PROGRAM MAIN
VAR
	RuntimeDuration	: STRING;
	TempRuntimeDur	: TIME;
	RuntimeTimer	: TON;
	CurrentSysTime	: ULINT;

	bAllDone		: BOOL;
	bStopSequence	: BOOL;
	HMI_StopCmd		: BOOL;
	
	nCase 		: INT;
	nMoveState		: ARRAY[1..nMoverCount] OF INT;
	

	
	nForCounter: UDINT;
	M,N,T,Tr : UINT;
//	slowDynamics: DynamicConstraint_PathXY;
	haltDynamics : DynamicConstraint_PathXY;
	stopAndWait : ARRAY[1..GVL_Mc.nMoverCount] OF TON; 
	waitForGapParkPos: LREAL := 3500;
	// Magnet
	MagnetValue AT%Q*: INT;
	MagnetFdbkValue AT%I* : INT;
	bMagnetOn : BOOL;
	MagnetOnManHMICmd 	: BOOL;
	tMagnetOnTime	: TIME := T#3S;

	Init : BOOL ; 	
	
	IsMoverCommandedInShortcut: BOOL;
	IsMoverInBlockingArea: BOOL;
	nActStopPos: UINT := 1;
	Fp_error : R_Trig;

	Switch : BOOL;
	WithoutSwitch : BOOL := TRUE;
	SwtichOnly: BOOL;
	
	MoverStop 	AT%I* :BOOL;
	MoverStopDone AT%Q*		: BOOL;
	Info 		AT%Q*: BOOL;
	Operating	AT%Q*: BOOL;
	Process		AT%Q*: BOOL;
	Fault		AT%Q*: BOOL;
	Emergency	AT%Q*: BOOL;
	
	Voltage1 AT%I*: UDINT;
	Voltage2 AT%I*: UDINT;
	
	
	TcRestart : TC_Restart;
	Restart : BOOL;
	busy : BOOL;
	rt_InitStart : R_TRIG;
	rt_InitStop : R_TRIG;
	bStartSequence: BOOL;
	
	FP_Counter : r_trig;
	Switchcounter : DINT;
	test : LREAL;
	Horntimer : tp; 
	R_trigHorn : R_trig;
	
	TestPowerMat : BOOL := TRUE;
	StopTime : TIME := T#1S;
	StopTimer :ARRAY[1..nMoverCount] OF ton;
	StartTimer :ARRAY[1..nMoverCount] OF BOOL;
	
	
	MoverPos :ARRAY[1..nMoverCount] OF PositionXYC;
	ArcLength :ARRAY[1..nMoverCount] OF LREAL;
	TrackPos :ARRAY[1..nMoverCount] OF ARRAY[1..nMoverCount] OF PositionXYC;
	
	//searchGap : F_SearchTheBigTrackForAHole; 
	aMoverTrack : ARRAY[1..nMoverCount] OF Global.OTCID;
	FirstMoverTrackPos : LREAL;
	MoverGap : LREAL;
	FTrigTrackCount : F_Trig;
	MoverNo  : UDINT;
	stMoverConfigSlow	: ST_MoverConfig;
	stMoverConfigNormal : ST_MoverConfig;
	stMoverConfigFast  : ST_MoverConfig;
	stMoverCfgAggressive : ST_MoverConfig;
	stMoverCfgHalt : ST_MoverConfig;
	
	stMergeConfig		 : ST_MergeConfig;
	SwitchConfig		 : ST_SwitchConfig;
	
	SwitchStatus 		  : ST_SwitchStatus;

	ModuleState1 AT%I*: E_EcState;
	ModuleState2 AT%I*: E_EcState;
	ModuleState3 AT%I*: ARRAY[0..2] OF E_EcState;
	
	MessageTrigger : ARRAY[1..20] OF R_trig;
	
	//========= Merge =========================================
	
	SwitchParkPos : LREAL := 3500;
	nextMoverForSwitch: UDINT :=1;
	moverInSwitchDoNotSendAnother: BOOL;
	trapError: BOOL;
	trapErrorID: UDINT;
	moverWithFault: UDINT;
	stepWithFault: INT;
	
	followSyncPos: LREAL;
	masterSyncPos: LREAL;
	masterPosAtSync: LREAL;
	followerPosAtSync: LREAL;
	moverInFront: UDINT;
	gapStart: LREAL := 8500; //5600
	gapLength: LREAL := 2200; //1800
	fbTrackobject : FB_TrackObject;
	getList: BOOL;
	directMerge: BOOL;
	mergeNotPossible: BOOL;
	
	endOfBigTrack : LREAL; 
	endOfSmallTrack : LREAL; 
	endOfMainTrack : LREAL; 
	followerToEndOfTrack: LREAL;
	leaderToEndofTrack: LREAL;
	distToMoverInFront: LREAL;
	moverSwitching: UDINT;
	switchingMoverPosition: LREAL;
	trapWhenMagnetturnedOn: R_TRIG;
	moverPositionWhenMagnetTurnedOn: LREAL;
	moverInSwitch: UDINT;
END_VAR


// =====================
// Initalize XTS Utility
GVL_MC.fbXtsEnvironment.Init(GVL_MC.cmdFeedback);
IF NOT GVL_MC.cmdFeedback.IsDone THEN
	RETURN;
END_IF
//*****************************************************
Emergency :=  MoverStop;

Operating := NOT  MoverStop;

//================== Check Voltage=====================================================
R_trigHorn(clk := Voltage1< 250000 );
//Horntimer(in:= ( R_trigHorn.Q ) , PT:= T#2S,Q=> info);
IF R_trigHorn.Q THEN
	ADSLOGSTR(msgCtrlMask:= ADSLOG_MSGTYPE_LOG , msgFmtStr:= 'Module Voltage Fault ' , strArg:= '');
END_IF 
//=================== Check State of Modules===========================================

MessageTrigger[1](clk:=ModuleState1 <> 8 AND nCASE> 0);
IF MessageTrigger[1].Q THEN
	ADSLOGSTR(msgCtrlMask:= ADSLOG_MSGTYPE_LOG , msgFmtStr:= 'Module Fault Line 1 %s' , strArg:= TO_STRING(ModuleState1));
END_IF

MessageTrigger[2](clk:=ModuleState2 <> 8 AND nCASE> 0);
IF MessageTrigger[2].Q THEN
	ADSLOGSTR(msgCtrlMask:= ADSLOG_MSGTYPE_LOG , msgFmtStr:= 'Module Fault Line 2 %s ' , strArg:= TO_STRING(ModuleState2));
END_IF

MessageTrigger[3](clk:=ModuleState3[0] <> 8 AND nCASE> 0);
IF MessageTrigger[3].Q THEN
	ADSLOGSTR(msgCtrlMask:= ADSLOG_MSGTYPE_LOG , msgFmtStr:= 'Module Fault Line 3 Default SyncUnit %s ' , strArg:= TO_STRING(ModuleState3[0]));
END_IF

MessageTrigger[4](clk:=ModuleState3[1] <> 8 AND nCASE> 0);
IF MessageTrigger[4].Q THEN
	ADSLOGSTR(msgCtrlMask:= ADSLOG_MSGTYPE_LOG , msgFmtStr:= 'Module Fault Line 3 XtsTask SyncUnit %s ' , strArg:= TO_STRING(ModuleState3[1]));
END_IF

MessageTrigger[5](clk:=ModuleState3[2] <> 8 AND nCASE> 0);
IF MessageTrigger[5].Q THEN
	ADSLOGSTR(msgCtrlMask:= ADSLOG_MSGTYPE_LOG , msgFmtStr:= 'Module Fault Line 3 PlcTask SyncUnit %s ' , strArg:= TO_STRING(ModuleState3[2]));
END_IF

//=====================================================================================

IF nCASE > 90 THEN
	Process := TRUE;
ELSE 
	Process := FALSE;	
END_IF

IF NOT MoverStop AND NOT MoverStopDone AND (nCase = 100) THEN
	ADSLOGSTR(msgCtrlMask:= ADSLOG_MSGTYPE_LOG , msgFmtStr:= 'E-Stop ' , strArg:= '');
	FOR nForCounter:=1 TO nNumMovers DO
		fbMover[nForCounter].P_Dynamics.SetValuesVADJ(stMoverConfigNormal.velo,stMoverConfigNormal.Accel,stMoverConfigNormal.Decel,stMoverConfigNormal.Jerk);
		nCase := 140;
	END_FOR		
ELSIF 	MoverStop THEN
	MoverStopDone := FALSE;
END_IF



TcRestart(
NETID:= '', 
RESTART:= Restart OR (GVL_Mc.HWStart AND NOT GVL_Mc.HWStop), 
TMOUT:=T#5S , 
BUSY=>busy , 
ERR=> , 
ERRID=> );

CurrentSysTime	:= Tc2_System.F_GetSystemTime();

IF TcRestart.BUSY THEN
	RuntimeTimer.IN 	:= FALSE;
ELSIF Process THEN
	RuntimeTimer.IN		:= TRUE;
	TempRuntimeDur		:= RuntimeTimer.ET;
	RuntimeDuration		:= TIME_TO_STRING(TempRuntimeDur);
END_IF
RuntimeTimer(PT := T#7D);

rt_InitStart(clk:= (bStartSequence OR GVL_Mc.HWStart) AND GVL_Mc.HWStop);
IF rt_InitStart.Q THEN
	nCase := 10;
	bStartSequence	:= FALSE;

	stMoverConfigSlow.Velo := 1000;
// 	stMoverConfigSlow.Accel := 4000;
// 	stMoverConfigSlow.Decel := 4000; 
// 	stMoverConfigSlow.Jerk := 16000;
	stMoverConfigFast.Velo := 4000;
// 	stMoverConfigFast.Accel := 4000;
// 	stMoverConfigFast.Decel := 4000; 
// 	stMoverConfigFast.Jerk := 16000;
	stMoverCfgHalt.Decel := 2000; 
	stMoverCfgHalt.Jerk := 10000;
	
//	slowDynamics.SetValuesVADJ(stMoverConfigSlow.Velo,stMoverConfigSlow.Accel,stMoverConfigSlow.Decel,stMoverConfigSlow.Jerk);
//	fastDynamics.SetValuesVADJ(stMoverConfigFast.Velo,stMoverConfigFast.Accel,stMoverConfigFast.Decel,stMoverConfigFast.Jerk);
	haltDynamics.SetValuesVADJ(stMoverCfgHalt.Velo,stMoverCfgHalt.Accel,stMoverCfgHalt.Decel,stMoverCfgHalt.Jerk);
END_IF
haltDynamics.SetValuesVADJ(stMoverCfgHalt.Velo,stMoverCfgHalt.Accel,stMoverCfgHalt.Decel,stMoverCfgHalt.Jerk);
GVL_Mc.StartLight := MoverStop AND nCase < 100;
GVL_Mc.StopLight  := (nCase = 100);

IsMoverInBlockingArea := FALSE;

FOR M := 1 TO GVL_Mc.nNumMovers DO///Movers
	StopTimer[M](in:=StartTimer[m],PT:=StopTime);

	
	IF NOT GVL_MC.fbMover[GVL_Mc.nNumMovers].P_IsInitialized THEN
		GVL_MC.ipXtsProcessingUnit :=  GVL_MC.fbXtsEnvironment.ProcessingUnit(1,0);
		GVL_MC.ipXlMover  :=  GVL_MC.fbXtsEnvironment.ProcessingUnit(1, 0).XlMover(m, 0);
		GVL_MC.fbMover[m].Init( GVL_MC.ipXlMover, GVL_MC.ipXtsProcessingUnit); 
		iMover[m] := fbMover[m] ;
	END_IF
	 MoverFeedback[m].Update();
	GVL_MC.fbMover[m].CycleUpdate();
	
	GVL_Mc.Mover[M].MoverPos  :=GVL_MC.fbMover[M].P_PlanarMover.MCTOPLC.SETONTRACK.SetPos;
	GVL_Mc.Mover[M].TrackID:= GVL_MC.fbMover[M].P_PlanarMover.MCTOPLC.SETONTRACK.TrackOID;
	GVL_Mc.Mover[M].MoverNumber := M;
		
	TR := Tr+1;
	IF Tr = 4 THEN
		Tr :=1;
	END_IF
	ArcLength[M] :=GVL_Mc.MC_Tracks[Tr].GetArcLengthClosestTo(MoverPos[M]);
	GVL_Mc.MC_Tracks[Tr].GetPositionAt(ArcLength[M],TrackPos[M][Tr]);
	
	IF ABS(MoverPos[m].x - TrackPos[M][Tr].x) < 1 AND  ABS(MoverPos[m].y - TrackPos[M][Tr].y) < 1 THEN
 		GVL_Mc.Mover[M].MoverTrackNr := Tr;
	END_IF	
	
	IsMoverInBlockingArea := IsMoverInBlockingArea OR (Mover[M].TrackID = GVL_Mc.MC_Tracks[E_TrackNum.main].MCTOPLC_STD.TrackOID AND IsBetween(Mover[M].MoverPos, SwitchConfig.MagnetStartPosition - 100, SwitchConfig.MagnetEndPosition + 100));

	Fp_error(clk := GVL_MC.fbMover[M].P_PlanarMover.Error AND GVL_MC.fbMover[M].XtsXlMover.GetIsActive(0) AND nCASE = 100);
	IF Fp_error.Q THEN
		nCase := 140;
		Fault := TRUE;
		bMagnetOn := FALSE;
		ADSLOGSTR(msgCtrlMask:= ADSLOG_MSGTYPE_LOG , msgFmtStr:= 'Mover %s Faulted ' , strArg:= INT_TO_STRING(M));
	ELSE
		Fault := FALSE;
	END_IF
	
	IF aMoverTrack[1] <> 0 AND_THEN GVL_MC.fbMover[M].P_PlanarMover.MCTOPLC.STD.MoverOID = aMoverTrack[1] THEN
		FirstMoverTrackPos := GVL_MC.fbMover[M].P_PlanarMover.MCTOPLC.SETONTRACK.SetPos;
	END_IF
	
END_FOR

FOR T := 1 TO nTrackCount DO 
	MC_Tracks[T].Update();
	MC_Trackfeedback[T].Update();
	
END_FOR
 MoverGap := (GVL_Mc.MC_Tracks[E_TrackNum.Big].GetLength()- FirstMoverTrackPos);
 
//================  merge ===============

fbTrackobject(TrackID:= MC_Tracks[E_TrackNum.big].MCTOPLC_STD.TrackOID,iMover:= iMover,trackLength:= GVL_Mc.MC_Tracks[E_TrackNum.Big].GetLength()); 
fbTrackobject.CyclicUpdate(); 


//======================================

CASE nCase OF
	10:
		
		Fault := FALSE;
		nCase := 20;

	20:
		FOR T := 1 TO nTrackCount DO 
			MC_Tracks[T].Enable(MC_Trackfeedback[T]);
		END_FOR
				nCase := 30;
				
	30: 
		IF MC_Trackfeedback[1].Done AND MC_Trackfeedback[2].Done AND MC_Trackfeedback[3].Done THEN
			nCase := 35;
		END_IF
		
		
	35:
		FOR nForCounter:=1 TO nNumMovers DO
			GVL_MC.fbMover[nForCounter].P_Dynamics.SetValuesVADJ(stMoverConfigNormal.velo,stMoverConfigNormal.Accel,stMoverConfigNormal.Decel,stMoverConfigNormal.Jerk);
			fbMover[nForCounter].P_PlanarMover.Reset(MoverFeedback[nForCounter]);
		END_FOR
		nCase := 36;	
			
	36:	
		bAllDone:=TRUE;
		FOR nForCounter:=1 TO nNumMovers DO
			bAllDone:=bAllDone AND MoverFeedback[nForCounter].Done;
		END_FOR
		
		IF bAllDone THEN
			nCase := 40;
		END_IF
				
	40:
		FOR nForCounter:=1 TO nNumMovers DO
			fbMover[nForCounter].P_PlanarMover.Enable(MoverFeedback[nForCounter]);
		END_FOR
		nCase := 50;
			
	50:
		bAllDone:=TRUE;
		FOR nForCounter:=1 TO nNumMovers DO
			bAllDone:=bAllDone AND MoverFeedback[nForCounter].Done;
		END_FOR
		
		IF bAllDone THEN
			nCase := 60;
		END_IF

	60:
		FOR nForCounter:=nNumMovers TO 1  BY -1 DO
			fbMover[nForCounter].JoinNearestTrack();
		END_FOR
		
		nCase := 70;
		
		
	70:
		bAllDone:=TRUE;
		FOR nForCounter:=1 TO nNumMovers DO
			bAllDone:=bAllDone AND fbMover[nForCounter].P_PlanarFeedback.Done;
		END_FOR
		
		IF bAllDone THEN
			nCase := 80;
		END_IF
		
	80:	
		FOR nForCounter:=1 TO nNumMovers DO
			nMoveState[nForCounter] := 0;
		END_FOR
		
		nCase := 100;

	100:
		
		FOR nForCounter:=1 TO nNumMovers DO
			fbMover[nForCounter].P_Dynamics.SetValuesVADJ(stMoverConfigNormal.velo,stMoverConfigNormal.Accel,stMoverConfigNormal.Decel,stMoverConfigNormal.Jerk);
			IF MoverNo <> 0 AND_THEN 	fbMover[MoverNo].P_PlanarMover.MCTOPLC.SETONTRACK.TrackOID =	 GVL_Mc.MC_Tracks[E_TrackNum.Big].MCTOPLC_STD.TrackOID THEN
				IsMoverCommandedInShortcut := FALSE;
			//	MoverNo := 0;
			END_IF
			
			//Adjust the first mover parameters to induce a platoon
			fbMover[1].P_Dynamics.SetValuesVADJ(V:= stMoverConfigNormal.velo-stMoverConfigNormal.VeloComp, A:= stMoverConfigNormal.Accel, D:= stMoverConfigNormal.Decel, J:= stMoverConfigNormal.Jerk);	
			
			IF SwitchConfig.DivertConfig.MaxAllowedDivertCount > 0 THEN
				WithoutSwitch 	:= FALSE;
			ELSE
				WithoutSwitch	:= TRUE;
			END_IF
			
			CASE nMoveState[nForCounter] OF
				
				0: // Track 3 Main Cycle
					fbMover[nForCounter].P_Dynamics.SetValuesVADJ(stMoverConfigNormal.velo,stMoverConfigNormal.Accel,stMoverConfigNormal.Decel,stMoverConfigNormal.Jerk);
					fbMover[nForCounter].MoveOnTrack(track:= GVL_Mc.MC_Tracks[E_TrackNum.Main], targetPos:= GVL_Mc.MC_Tracks[E_TrackNum.Main].GetLength()-500, gap:= stMoverConfigNormal.MoverGap);
				
					nMoveState[nForCounter] := 10;
					
				10:
					IF Mover[nForCounter].MoverPos > GVL_Mc.MC_Tracks[E_TrackNum.Main].GetLength()-6000  AND  Mover[nForCounter].TrackID =   GVL_Mc.MC_Tracks[E_TrackNum.Main].MCTOPLC_STD.TrackOID    THEN//     MCTrackOid_MainSemicircle THEN
						IF  (SwtichOnly OR NOT IsMoverCommandedInShortcut )AND NOT WithoutSwitch  AND  nForCounter = nextMoverForSwitch THEN // AND NOT( moverInSwitchDoNotSendAnother)  THEN
							nMoveState[nForCounter] := 40; // 20 - BigCycel
								moverInSwitchDoNotSendAnother := TRUE; 
							//IF fbPlanarMover[nForCounter].IsCommandedInShortcut THEN
								IsMoverCommandedInShortcut := TRUE;
								MoverNo :=nForCounter; /// fbPlanarMover[nForCounter].McPlanarMover.MCTOPLC.STD.MoverOID;
								IF nextMoverForSwitch >= nNumMovers THEN // send the next mover to the switch
									nextMoverForSwitch := 1; 
								ELSE 
									nextMoverForSwitch := nextMoverForSwitch + 1; 
								END_IF
							//END_IF
						ELSE
							nMoveState[nForCounter] := 20;  // 40- SmallCycel					
						END_IF
					END_IF

				
				20:
					fbMover[nForCounter].P_Dynamics.SetValuesVADJ(stMoverConfigNormal.velo,stMoverConfigNormal.Accel,stMoverConfigNormal.Decel,stMoverConfigNormal.Jerk);
					fbMover[nForCounter].MoveOnTrack(track:= GVL_Mc.MC_Tracks[E_TrackNum.Big], targetPos:= GVL_Mc.MC_Tracks[E_TrackNum.Big].GetLength()-1000, gap:= stMoverConfigNormal.MoverGap);
			
					nMoveState[nForCounter] := 30;
				
					
				30:
					IF fbMover[nForCounter].P_PlanarFeedback.Error AND NOT trapError THEN //trap the error once.  
						moverWithFault := nForCounter; 
						trapError := fbMover[nForCounter].P_PlanarFeedback.Error; 
						trapErrorID := fbMover[nForCounter].P_PlanarFeedback.ErrorId; 
						stepWithFault := 30; 
					END_IF 
					IF Mover[nForCounter].MoverPos > GVL_Mc.MC_Tracks[E_TrackNum.Big].GetLength()-12000 AND  Mover[nForCounter].TrackID = GVL_Mc.MC_Tracks[E_TrackNum.big].MCTOPLC_STD.TrackOID    THEN//      MCTrackOid_BigSemicircle THEN
						nMoveState[nForCounter] := 0;
					END_IF				
				
			
				40:
					fbMover[nForCounter].P_Dynamics.SetValuesVADJ(stMoverConfigNormal.velo,stMoverConfigNormal.Accel,stMoverConfigNormal.Decel,stMoverConfigNormal.Jerk);
					fbMover[nForCounter].MoveOnTrack(track:= GVL_Mc.MC_Tracks[E_TrackNum.Small], targetPos:= SwitchParkPos, gap:= stMoverConfigNormal.MoverGap);
					
					nMoveState[nForCounter] := 45;
	
				45: 
					IF fbMover[nForCounter].P_PlanarFeedback.Error AND NOT trapError THEN //trap the error once.   
						trapError := fbMover[nForCounter].P_PlanarFeedback.Error; 
						trapErrorID := fbMover[nForCounter].P_PlanarFeedback.ErrorId;
						stepWithFault := 45;
 						moverWithFault := nForCounter; 
					END_IF
					IF fbMover[nForCounter].P_PlanarFeedback.Done THEN 
						nMoveState[nForCounter] := 50; //50;
						stopAndWait[nForCounter](IN:=TRUE, PT:=StopTime); 
					END_IF 	

				50:
					stopAndWait[nForCounter](); 
					IF stopAndWait[nForCounter].Q  OR NOT TestPowerMat THEN // send the mover to a sync Position 2.6m before the end of the track 
						stopAndWait[nForCounter](IN:=FALSE); 							
					//	fbMover[nForCounter].P_Dynamics.SetValuesVADJ(stMoverConfigNormal.velo,stMoverConfigNormal.Accel,stMoverConfigNormal.Decel,stMoverConfigNormal.Jerk);
					//	fbMover[nForCounter].MoveOnTrack( GVL_Mc.MC_Tracks[E_TrackNum.Small], GVL_Mc.MC_Tracks[E_TrackNum.Small].GetLength()-waitForGapParkPos,stMoverConfigNormal.MoverGap,stMoverConfigNormal.velo);
					//	searchGap(resetSearch:=TRUE, fbMover := fbMover); 
						nMoveState[nForCounter] := 60; 
					END_IF 
					
				60: // look for a merge position 
					//IF fbMover[nForCounter].P_PlanarFeedback.Done THEN// MCTrackOid_Shortcut THEN
							fbTrackobject.findMergePosition(
								mergeSyncCommandPos := gapStart , 
								spaceToMerge := gapLength, 
								nMoverToFollow => moverInFront, 
								mergeWithoutFollow => directMerge, 
								mergeNotPossible => mergeNotPossible); 
							IF directMerge OR  ( moverInFront <> 0) AND NOT mergeNotPossible THEN
								nMoveState[nForCounter] := 70;
							END_IF 
				//	END_IF
				70:  //merge with gap zero
					//issue commmand to sync 
					IF  directMerge THEN 
						fbMover[nForCounter].P_Dynamics.SetValuesVADJ(stMoverConfigNormal.velo,stMoverConfigNormal.Accel,stMoverConfigNormal.Decel,stMoverConfigNormal.Jerk);
						fbMover[nForCounter].MoveOnTrack(track:= GVL_Mc.MC_Tracks[E_TrackNum.Main], targetPos:= GVL_Mc.MC_Tracks[E_TrackNum.Main].GetLength()-500, gap:= stMoverConfigNormal.MoverGap);

						nMoveState[nForCounter] := 10; 
					ELSIF moverInFront <>0 THEN 
						fbMover[nForCounter].P_Dynamics.SetValuesVADJ(stMoverConfigNormal.velo,stMoverConfigNormal.Accel,stMoverConfigNormal.Decel,stMoverConfigNormal.Jerk);
						masterSyncPos := GVL_Mc.MC_Tracks[E_TrackNum.Big].GetLength()-2500;
						masterPosAtSync := Mover[moverInFront].MoverPos; 
						followSyncPos := GVL_Mc.MC_Tracks[E_TrackNum.Small].GetLength()-stMoverConfigNormal.MoverGap-2500;
						followerPosAtSync :=Mover[nForCounter].MoverPos; 
						fbMover[nForCounter].SyncToOtherMover( 
							masterSyncPos := masterSyncPos,
							masterTrack := GVL_Mc.MC_Tracks[E_TrackNum.Big],
							followerSyncPos := followSyncPos,
							followerTrack := GVL_Mc.MC_Tracks[e_TrackNum.Small],
							PlanarMoverToFollow := fbMover[moverInFront].P_PlanarMover,
							velo:= stMoverConfigNormal.velo);
							nMoveState[nForCounter] := 80; 
						// reduce the gap of the leading mover 
						fbMover[moverInFront].MoveOnTrack(track:= GVL_Mc.MC_Tracks[E_TrackNum.Main], targetPos:= GVL_Mc.MC_Tracks[E_TrackNum.Main].GetLength()-500, gap:= 0);

					END_IF 
					
				80: // wait for in Sync 
					IF fbMover[nForCounter].P_SyncFeedback.Active AND MOver[moverInFront].TrackID =  GVL_Mc.MC_Tracks[E_TrackNum.Big].MCTOPLC_STD.TrackOID THEN // actively syncing calculate distance from mover 
						followerToEndOfTrack := fbMover[nForCounter].distToEndOfTrack; 
						leaderToEndofTrack := fbMover[moverInFront].distToEndOfTrack; 
						distToMoverInFront := followerToEndOfTrack - leaderToEndofTrack; 
					ELSE 
						followerToEndOfTrack := 0; 
						leaderToEndofTrack := 0; 
						distToMoverInFront := 0;
					END_IF
					IF fbMover[nForCounter].P_SyncFeedback.inSync OR  MOver[nForCounter].TrackID =  GVL_Mc.MC_Tracks[E_TrackNum.Main].MCTOPLC_STD.TrackOID THEN 
						nMoveState[nForCounter] := 10;
						IsMoverCommandedInShortcut :=FALSE;
					ELSIF	fbMover[nForCounter].P_SyncFeedback.Error THEN
						nMoveState[nForCounter] := 60;
					END_IF 
					
				END_CASE
		
		END_FOR

		rt_InitStop(CLK := HMI_StopCmd OR NOT GVL_Mc.HWStop);
		IF rt_InitStop.Q AND NOT bStopSequence THEN
			bStopSequence := TRUE;
		END_IF
		IF bStopSequence AND NOT(IsMoverInBlockingArea) THEN
			nCase := 110;
			bStopSequence := FALSE;
		END_IF
		
		110:
			N:= nNumMovers;
			FOR nForCounter:=1 TO nNumMovers DO		
				aStopPositions[nForCounter] := fbMover[nForCounter].XtsXlMover.GetSimulatedStartUpPosition(0);
				N := N -1;
			END_FOR
			nCase := 120;
		
		120:	
			nActStopPos := UDINT_TO_UINT(nMoverCount-nNumMovers+1);
			FOR nForCounter:=1 TO nNumMovers DO
				fbMover[nForCounter].P_Dynamics.SetValuesVADJ(stMoverConfigNormal.velo,stMoverConfigNormal.Accel,stMoverConfigNormal.Decel,stMoverConfigNormal.Jerk);
				nMoveState[nForCounter] := 0;
				fbMover[nForCounter].MoveOnTrack(track:= GVL_Mc.MC_Tracks[E_TrackNum.Main], targetPos:= 300, gap:= stMoverConfigNormal.MoverGap);
			END_FOR

			nCase:= 130; 
		130:
			FOR nForCounter:=1 TO nMoverCount - (nMoverCount -nNumMovers)  DO
				CASE nMoveState[nForCounter] OF
					0:								
						IF Mover[nForCounter].MoverPos < 300 AND  Mover[nForCounter].TrackID = GVL_Mc.MC_Tracks[E_TrackNum.main].MCTOPLC_STD.TrackOID THEN
							fbMover[nForCounter].MoveOnTrack(track:= GVL_Mc.MC_Tracks[E_TrackNum.Main], targetPos:= aStopPositions[nActStopPos], gap:= stMoverConfigNormal.MoverGap);

							nActStopPos := nActStopPos + 1;
							nMoveState[nForCounter] := 10;
						END_IF
				END_CASE
			END_FOR
		
			bAllDone := TRUE;
			FOR nForCounter:=1 TO nNumMovers DO
				IF NOT(MoverFeedback[nForCounter].Done OR MoverFeedback[nForCounter].Error) THEN
					bAllDone := FALSE;
					EXIT;
				END_IF
			END_FOR
			
			IF bAllDone THEN
				nCase := 150;
			END_IF
		
		140:
			FOR nForCounter:=1 TO nNumMovers DO
				fbMover[nForCounter].P_PlanarMover.Halt(MoverFeedback[nForCounter], haltDynamics);
			END_FOR	
			
		nCase := 145;
			
		145:
			bAllDone := TRUE;
			FOR nForCounter:=1 TO nNumMovers DO
				IF NOT(MoverFeedback[nForCounter].Done OR MoverFeedback[nForCounter].Error) THEN
					bAllDone := FALSE;
					EXIT;
				END_IF
			END_FOR
			
			IF bAllDone THEN
				nCase := 150;
			END_IF
		
		//Disable
		150:

			FOR nForCounter:=1 TO nNumMovers DO
				fbMover[nForCounter].P_PlanarMover.Disable(MoverFeedback[nForCounter]);
			END_FOR
				
			nCase := 155;
		155:
			bAllDone := TRUE;
			FOR nForCounter:=1 TO nNumMovers DO
				IF NOT(MoverFeedback[nForCounter].Done OR MoverFeedback[nForCounter].Error) THEN
					bAllDone := FALSE;
					EXIT;
				END_IF
			END_FOR
			
			IF bAllDone THEN
				//MoverStopDone := TRUE;
				nCase := 0;
			END_IF	
END_CASE

bMagnetOn := FALSE;
FOR nForCounter:=1 TO nNumMovers DO
	IF  fbMover[nForCounter].XtsXlMover.GetPositionInfo_trackObjectId(0) = XtsShortcutOid THEN // this mover wll go through the switch start tracking his positon 
		switchingMoverPosition := fbMover[nForCounter].XtsXlMover.GetPositionInfo_trackPosition(0);  
	END_IF
	// check if the mover is in range of the switch position and on the switch track, if so turn on the magnet 
	IF fbMover[nForCounter].XtsXlMover.GetPositionInfo_trackObjectId(0) = XtsShortcutOid AND (IsBetween(fbMover[nForCounter].XtsXlMover.GetPositionInfo_trackPosition(0), SwitchConfig.MagnetStartPosition - (stMoverConfigNormal.Velo*0.045), SwitchConfig.MagnetEndPosition)) THEN
		bMagnetOn := TRUE; 
	END_IF
	moverInSwitch := nForCounter; 
END_FOR


IF SwitchConfig.UseNominalCurrentVeloSetpoints THEN
	SwitchStatus.CurrentTheorOutputMax := SwitchConfig.SwitchCurrentNominal;	
ELSE
	SwitchStatus.CurrentTheorOutputMax := ((SwitchConfig.DivertConfig.CurrentFunctionCoeffA*(((stMoverConfigNormal.Velo/1000)*(stMoverConfigNormal.Velo/1000))))+(SwitchConfig.DivertConfig.CurrentFunctionCoeffB*(stMoverConfigNormal.Velo/1000))+SwitchConfig.DivertConfig.CurrentFunctionCoeffC);	
END_IF

SwitchStatus.CurrentActualOutput := F_MapLReal(
	x:= MagnetFdbkValue, 
	in_min:= 0, 
	in_max:= 32767, 
	out_min:= 0, 
	out_max:= 54);

IF (nCase = 100) THEN
	IF bMagnetOn AND NOT Fault THEN
		MagnetValue := TO_INT(SwitchStatus.CurrentTheorOutputMax*1310);
	ELSE
		MagnetValue := 0;
	END_IF
ELSE // Manual Control of the Magnet Coil
	IF MagnetOnManHMICmd THEN
		MagnetValue := TO_INT(SwitchStatus.CurrentTheorOutputMax*1310);
	ELSE
		MagnetValue := 0;
		MagnetOnManHMICmd	:= FALSE;
	END_IF
END_IF


trapWhenMagnetturnedOn(CLK:= bMagnetOn); 
IF moverInSwitch <> 0 AND trapWhenMagnetTurnedOn.Q THEN 
	moverPositionWhenMagnetTurnedOn:=fbMover[moverInSwitch].XtsXlMover.GetPositionInfo_trackPosition(0);
END_IF


FP_Counter(clk:=bMagnetOn);

IF FP_Counter.Q THEN
	Switchcounter := Switchcounter+1;

END_IF



//distanceMonitoring of Mover 1 when on the big track 
IF Mover[1].TrackID = GVL_Mc.MC_Tracks[E_TrackNum.Main].MCTOPLC_STD.TrackOID THEN //calculate out how far it is to the mover in front 
	IF MOver[stMergeConfig.moverInFront].MoverPos -  Mover[1].MoverPos > 10 THEN 
		stMergeConfig.mover1FollowDist := MOver[stMergeConfig.moverInFront].MoverPos -  Mover[1].MoverPos;
	END_IF   
END_IF

END_PROGRAM

(* stored: Version 1.1.0.1, ProductVersion 3.1.4026.8
   POU MAIN: Id {741d33e8-52ed-4b62-8ea9-8d206e7291c9}, SpecialFunc None *)
